PROGRAM PRG_VfdModbusRtu
VAR
	fbVfdMb: ModbusRtuMaster_KL6x22B;
	fbRTrigWrite: R_TRIG;
	fbRTrigEnable: R_TRIG;
	fbRTrigDisable: R_TRIG;
	fbRTrigReverseMotor: R_TRIG;
	fbRTrigSetFrequency: R_TRIG;
	fbTON: TON;
	fbTON1: TON;
	fbTON2: TON;
	fbTON3: TON;
	wQty: WORD := 1;
	wMbAddr: WORD;
	wCmd: WORD;
	wCmdPrev: WORD;
	bWrite: BOOL;
	bEnablePulse: BOOL;
	bPendingFlag: BOOL;
	bPulse: BOOL;
	bSetFreqCmd: BOOL;
	nSetFreqState: INT;
	nSetFreqVal: WORD;
END_VAR

fbRTrigWrite(CLK:=bWrite, Q=>);
fbRTrigEnable(CLK:= GVL.bRunVfd OR GVL.bEnable, Q=>);
fbRTrigDisable(CLK:= GVL.bStopVfd OR GVL.bDisable, Q=>);
fbRTrigReverseMotor(CLK:= GVL.bReverseMotor, Q=> );
fbRTrigSetFrequency(CLK:= GVL.bSetMotorFrequency, Q=> );

//Enable control word
IF fbRTrigEnable.Q THEN
	IF bWrite THEN
		bPendingFlag := TRUE; //Raise flag for pending command
	ELSE
		bWrite := TRUE;
	END_IF
	bEnablePulse := TRUE;
	wMbAddr := 417;
	wCmd := 32771;
END_IF

//Disable control word
IF fbRTrigDisable.Q THEN
	IF bWrite THEN
		bPendingFlag := TRUE; //Raise flag for pending command
	ELSE
		bWrite := TRUE;
	END_IF
	
	bEnablePulse := FALSE;
	wMbAddr := 417;
	wCmd := 0;
END_IF

//Reverse motor
IF fbRTrigReverseMotor.Q THEN
	IF bWrite THEN
		bPendingFlag := TRUE; //Raise flag for pending command
	ELSE
		bWrite := TRUE;
	END_IF
	bEnablePulse := TRUE;
	wMbAddr := 417;
	wCmd := 32777;	
END_IF

//Set motor frequency
IF fbRTrigSetFrequency.Q THEN
	bSetFreqCmd := TRUE;
	wCmdPrev := wCmd;
END_IF

IF bSetFreqCmd THEN
	CASE nSetFreqState OF
		0: //Set frequency
			IF bWrite THEN
				bPendingFlag := TRUE; //Raise flag for pending command
			ELSE
				bWrite := TRUE;
			END_IF
			bEnablePulse := FALSE;
			wMbAddr := 215;
			wCmd := nSetFreqVal*10;
			IF fbVfdMb.BUSY THEN
				nSetFreqState := 1;
			END_IF
		1: //Continue the previous command
			bSetFreqCmd := FALSE;
			IF wCmdPrev <> 0 THEN
				bEnablePulse := TRUE; //Short delay before pulse starts
				wMbAddr := 417;
				wCmd := wCmdPrev;
			END_IF
			nSetFreqState := 0;
	END_CASE
END_IF
//Keep sending enable signal to avoid watchdog error
fbTON1(IN:= bEnablePulse AND NOT fbTON2.Q, PT:= T#600MS, Q=> bPulse, ET=> ); //Pulse off time
fbTON2(IN:= fbTON1.Q, PT:= T#300MS, Q=> , ET=> );//Pulse on time

CASE wCmd OF
	32771: //Run motor forward
		GVL.bEnable := bPulse;
	32777: //Reverse motor
		GVL.bReverseMotor := bPulse;
END_CASE

IF bWrite THEN
	fbTON(IN:= bWrite, PT:= T#100MS, Q=> , ET=> );
END_IF

//Reset bWrite after a short delay
IF fbTON.Q THEN
	fbTON(IN:=FALSE);
	bWrite := FALSE;
END_IF

//Handle the raised pending flag
IF bPendingFlag AND NOT bWrite THEN
	fbTON3(IN:= TRUE, PT:= T#100MS, Q=> , ET=> );
END_IF

IF fbTON3.Q THEN
	fbTON3(IN:= FALSE);
	bPendingFlag := FALSE;
	bWrite := TRUE;
END_IF

fbVfdMb.WriteRegs(
	UnitID:= 1, 
	Quantity:= wQty, 
	MBAddr:= wMbAddr, 
	cbLength:= SIZEOF(wCmd), 
	pMemoryAddr:= ADR(wCmd), 
	Execute:= bWrite,//fbRTrigWrite.Q, 
	Timeout:= T#1S, 
	BUSY=> , 
	Error=> , 
	ErrorId=> , 
	cbRead=> );

END_PROGRAM

(* stored: Version 1.1.0.1, ProductVersion 3.1.4024.12
   POU PRG_VfdModbusRtu: Id {9519abab-4381-406c-81bf-d5d84071b90e}, SpecialFunc None *)
